FUNCTION_BLOCK FB_PosNear
VAR_INPUT
	AxisIdx		: INT;
	Offset		: LREAL;
END_VAR
VAR_OUTPUT
	IsNear		: BOOL:=FALSE;
END_VAR
VAR
	ActPos		: LREAL;
	SetPos		: LREAL;
	ActMSet		: LREAL;
	OffsetByCount: LREAL;
	Scaling		: LREAL:=1;
END_VAR

IsNear			 := FALSE;
ActPos			 := Axis[AxisIdx].Axis.NcToPlc.ActPos;
SetPos			 := Axis[AxisIdx].Axis.NcToPlc.SetPos;
ActMSet			 := ABS(ActPos - SetPos);
OffsetByCount	 := Offset*Scaling;
IF  ActMSet <= OffsetByCount THEN
	IsNear	:= TRUE;
END_IF

END_FUNCTION_BLOCK

(* stored: Version 1.1.0.1, ProductVersion 3.1.4024.9
   POU FB_PosNear: Id {a1051348-cece-4d80-a5bb-f772a230f4ba}, SpecialFunc None *)
